// TIA Portal V15.1 export
// export: Created 2024-05-17T05:38:27.7675341Z, ExportSetting WithDefaults, DisplayName Totally Integrated Automation Portal, DisplayVersion V15.1 Update 5, DisplayName TIA Portal Openness, DisplayVersion V15.1 Update 5, DisplayName SINAMICS Startdrive Advanced, DisplayVersion V15.1, DisplayName G130, G150, S120, S150, SINAMICS MV, S210, DisplayVersion V15.1, DisplayName G110M, G120, G120C, G120D, G120P, DisplayVersion V15.1, DisplayName STEP 7 Professional, DisplayVersion V15.1 Update 5, DisplayName STEP 7 Safety, DisplayVersion V15.1, DisplayName WinCC Professional, DisplayVersion V15.1 Update 5, DisplayName SIMATIC Visualization Architect, DisplayVersion V15.1
FUNCTION "CommStnS7Sv" : Void   // FC1900, FBD
TITLE = CommStnS7Sv
{ S7_Optimized_Access := 'TRUE' }
VERSION : 0.1
// This FC sends and receives data from and to the supervision.
// stored: AutoNumber false, IsIECCheckEnabled false, SetENOAutomatically False, UDAEnableTagReadback false
   VAR_INPUT
      PlcActiveShift : Int;
      PlcActiveBreak : Int;
      AlarmA : Bool;
      AlarmB : Bool;
      AlarmC : Bool;
      AlarmD : Bool;
      ModeAutoStep : Bool;
      ModeAutoSel : Bool;
      ModeMan : Bool;
      ModeManSel : Bool;
      StnAux01Feedback_Int : Int;
      StnAux02Feedback_Int : Int;
      StnAux03Feedback_Int : Int;
      StnAux04Feedback_Int : Int;
      StnAux05Feedback_Int : Int;
      StnAux06Feedback_Int : Int;
      StnAux07Feedback_DInt : DInt;
      StnAux08Feedback_DInt : DInt;
      StnAux09Feedback_DInt : DInt;
      StnAux10Feedback_DInt : DInt;
      StnAux11Feedback_DInt : DInt;
      StnAux12Feedback_DInt : DInt;
      StnAux13Feedback_Real : Real;
      StnAux14Feedback_Real : Real;
      StnAux15Feedback_Real : Real;
      StnAux16Feedback_Real : Real;
      StnAux17Feedback_Real : Real;
      StnAux18Feedback_Real : Real;
   END_VAR
   VAR_IN_OUT
      DB_ZMToSv : "SupervisionZM";   // Send to supervision system
      DB_SvToZM : "SupervisionZM";   // Recieve from supervision system
   END_VAR
   VAR_TEMP
      Tmp_StnAux13Feedback_Real : Real;
      Tmp_StnAux14Feedback_Real : Real;
      Tmp_StnAux15Feedback_Real : Real;
      Tmp_StnAux16Feedback_Real : Real;
      Tmp_StnAux17Feedback_Real : Real;
      Tmp_StnAux18Feedback_Real : Real;
   END_VAR
BEGIN

REGION Network 1: **** 8 - Outputs **** Plc ActiveShift
   // Plc ActiveShift
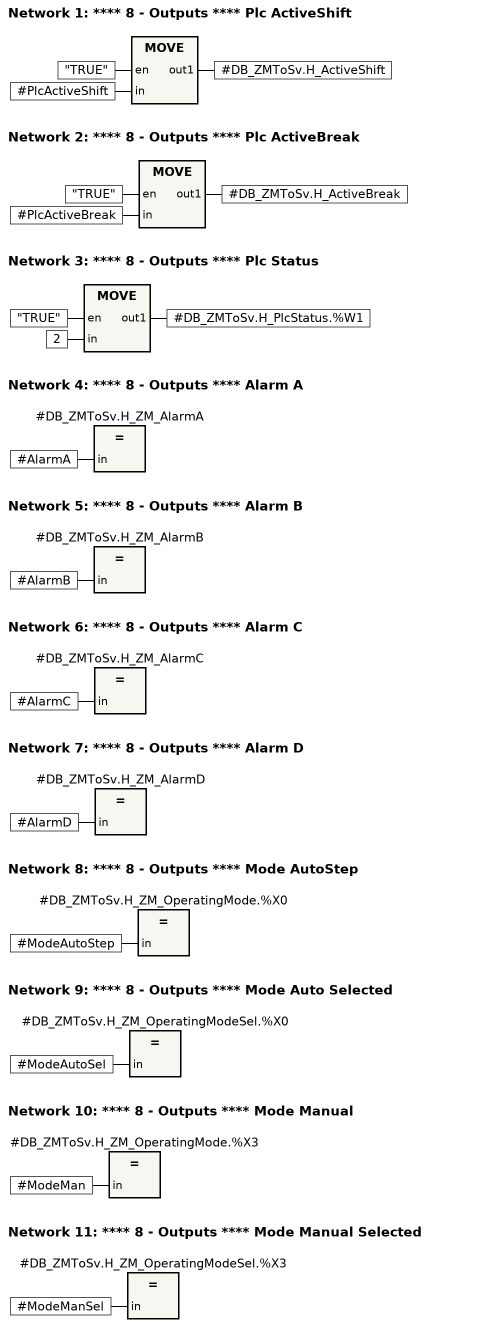
   IF "TRUE" THEN #DB_ZMToSv.H_ActiveShift := #PlcActiveShift; END_IF;
END_REGION

REGION Network 2: **** 8 - Outputs **** Plc ActiveBreak
   // Plc ActiveBreak
   IF "TRUE" THEN #DB_ZMToSv.H_ActiveBreak := #PlcActiveBreak; END_IF;
END_REGION

REGION Network 3: **** 8 - Outputs **** Plc Status
   // Plc Status
   IF "TRUE" THEN #DB_ZMToSv.H_PlcStatus.%W1 := 2; END_IF;
END_REGION

REGION Network 4: **** 8 - Outputs **** Alarm A
   // Alarm A
   #DB_ZMToSv.H_ZM_AlarmA := #AlarmA;
END_REGION

REGION Network 5: **** 8 - Outputs **** Alarm B
   // Alarm B
   #DB_ZMToSv.H_ZM_AlarmB := #AlarmB;
END_REGION

REGION Network 6: **** 8 - Outputs **** Alarm C
   // Alarm C
   #DB_ZMToSv.H_ZM_AlarmC := #AlarmC;
END_REGION

REGION Network 7: **** 8 - Outputs **** Alarm D
   // Alarm D
   #DB_ZMToSv.H_ZM_AlarmD := #AlarmD;
END_REGION

REGION Network 8: **** 8 - Outputs **** Mode AutoStep
   // Mode AutoStep
   #DB_ZMToSv.H_ZM_OperatingMode.%X0 := #ModeAutoStep;
END_REGION

REGION Network 9: **** 8 - Outputs **** Mode Auto Selected
   // Mode Auto Selected
   #DB_ZMToSv.H_ZM_OperatingModeSel.%X0 := #ModeAutoSel;
END_REGION

REGION Network 10: **** 8 - Outputs **** Mode Manual
   // Mode Manual
   #DB_ZMToSv.H_ZM_OperatingMode.%X3 := #ModeMan;
END_REGION

REGION Network 11: **** 8 - Outputs **** Mode Manual Selected
   // Mode Manual Selected
   #DB_ZMToSv.H_ZM_OperatingModeSel.%X3 := #ModeManSel;
END_REGION

REGION Network 12: **** 8 - Outputs **** Station Aux 01 Feedback
   // Station Aux 01 Feedback
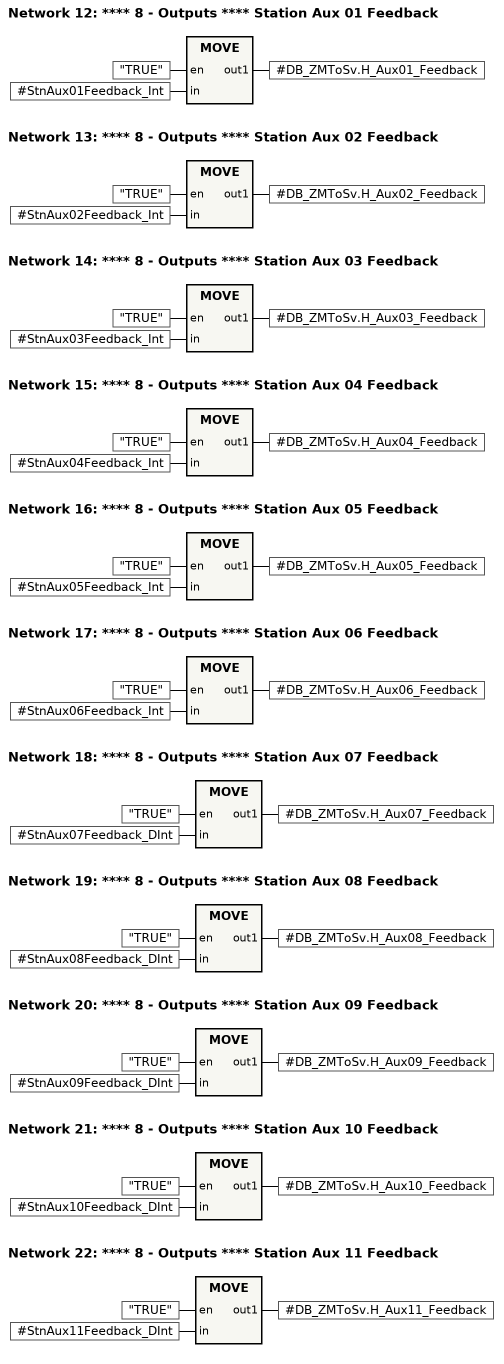
   IF "TRUE" THEN #DB_ZMToSv.H_Aux01_Feedback := #StnAux01Feedback_Int; END_IF;
END_REGION

REGION Network 13: **** 8 - Outputs **** Station Aux 02 Feedback
   // Station Aux 02 Feedback
   IF "TRUE" THEN #DB_ZMToSv.H_Aux02_Feedback := #StnAux02Feedback_Int; END_IF;
END_REGION

REGION Network 14: **** 8 - Outputs **** Station Aux 03 Feedback
   // Station Aux 03 Feedback
   IF "TRUE" THEN #DB_ZMToSv.H_Aux03_Feedback := #StnAux03Feedback_Int; END_IF;
END_REGION

REGION Network 15: **** 8 - Outputs **** Station Aux 04 Feedback
   // Station Aux 04 Feedback
   IF "TRUE" THEN #DB_ZMToSv.H_Aux04_Feedback := #StnAux04Feedback_Int; END_IF;
END_REGION

REGION Network 16: **** 8 - Outputs **** Station Aux 05 Feedback
   // Station Aux 05 Feedback
   IF "TRUE" THEN #DB_ZMToSv.H_Aux05_Feedback := #StnAux05Feedback_Int; END_IF;
END_REGION

REGION Network 17: **** 8 - Outputs **** Station Aux 06 Feedback
   // Station Aux 06 Feedback
   IF "TRUE" THEN #DB_ZMToSv.H_Aux06_Feedback := #StnAux06Feedback_Int; END_IF;
END_REGION

REGION Network 18: **** 8 - Outputs **** Station Aux 07 Feedback
   // Station Aux 07 Feedback
   IF "TRUE" THEN #DB_ZMToSv.H_Aux07_Feedback := #StnAux07Feedback_DInt; END_IF;
END_REGION

REGION Network 19: **** 8 - Outputs **** Station Aux 08 Feedback
   // Station Aux 08 Feedback
   IF "TRUE" THEN #DB_ZMToSv.H_Aux08_Feedback := #StnAux08Feedback_DInt; END_IF;
END_REGION

REGION Network 20: **** 8 - Outputs **** Station Aux 09 Feedback
   // Station Aux 09 Feedback
   IF "TRUE" THEN #DB_ZMToSv.H_Aux09_Feedback := #StnAux09Feedback_DInt; END_IF;
END_REGION

REGION Network 21: **** 8 - Outputs **** Station Aux 10 Feedback
   // Station Aux 10 Feedback
   IF "TRUE" THEN #DB_ZMToSv.H_Aux10_Feedback := #StnAux10Feedback_DInt; END_IF;
END_REGION

REGION Network 22: **** 8 - Outputs **** Station Aux 11 Feedback
   // Station Aux 11 Feedback
   IF "TRUE" THEN #DB_ZMToSv.H_Aux11_Feedback := #StnAux11Feedback_DInt; END_IF;
END_REGION

REGION Network 23: **** 8 - Outputs **** Station Aux 12 Feedback
   // Station Aux 12 Feedback
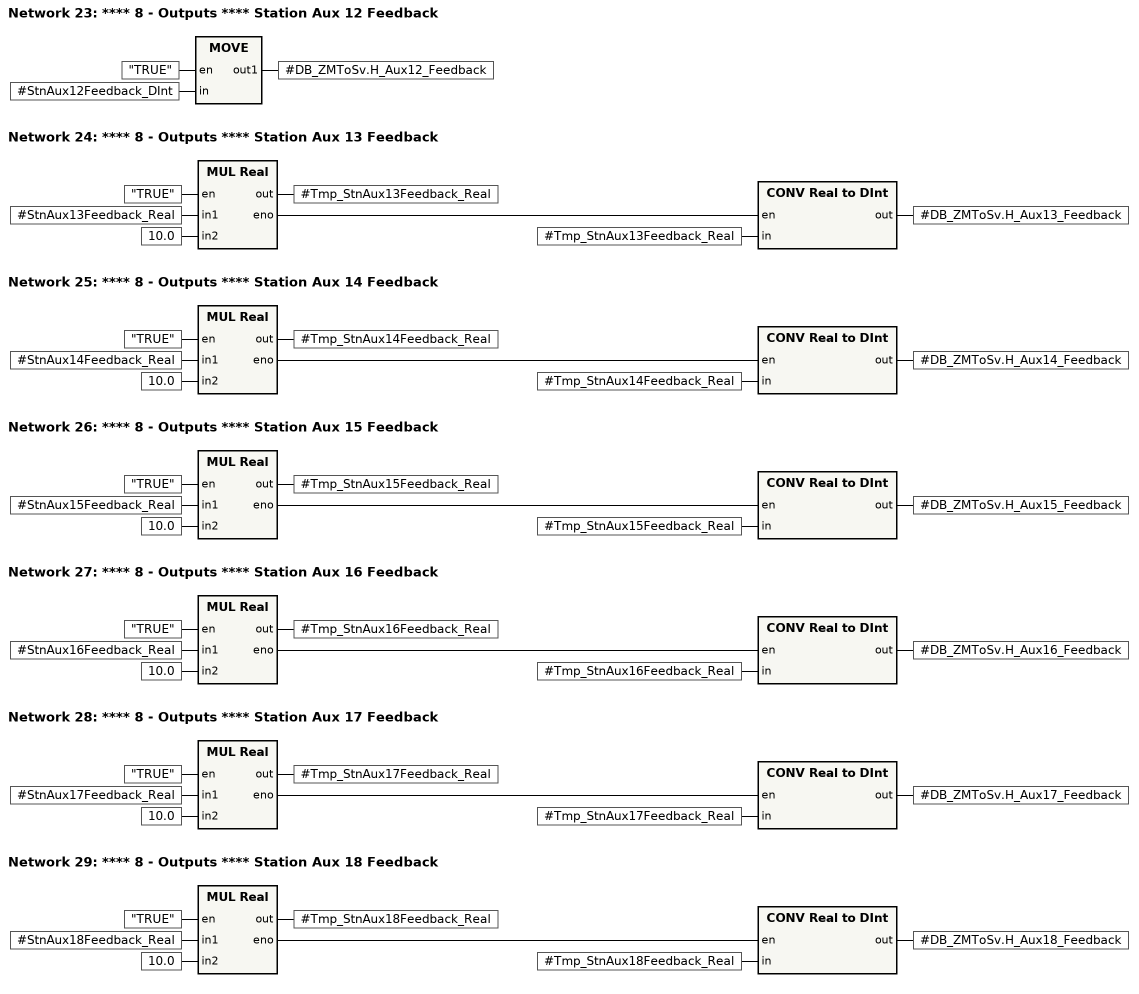
   IF "TRUE" THEN #DB_ZMToSv.H_Aux12_Feedback := #StnAux12Feedback_DInt; END_IF;
END_REGION

REGION Network 24: **** 8 - Outputs **** Station Aux 13 Feedback
   // Station Aux 13 Feedback
   IF "TRUE" THEN
       #Tmp_StnAux13Feedback_Real := #StnAux13Feedback_Real * 10.0;
       #DB_ZMToSv.H_Aux13_Feedback := REAL_TO_DINT(#Tmp_StnAux13Feedback_Real);
   END_IF;
END_REGION

REGION Network 25: **** 8 - Outputs **** Station Aux 14 Feedback
   // Station Aux 14 Feedback
   IF "TRUE" THEN
       #Tmp_StnAux14Feedback_Real := #StnAux14Feedback_Real * 10.0;
       #DB_ZMToSv.H_Aux14_Feedback := REAL_TO_DINT(#Tmp_StnAux14Feedback_Real);
   END_IF;
END_REGION

REGION Network 26: **** 8 - Outputs **** Station Aux 15 Feedback
   // Station Aux 15 Feedback
   IF "TRUE" THEN
       #Tmp_StnAux15Feedback_Real := #StnAux15Feedback_Real * 10.0;
       #DB_ZMToSv.H_Aux15_Feedback := REAL_TO_DINT(#Tmp_StnAux15Feedback_Real);
   END_IF;
END_REGION

REGION Network 27: **** 8 - Outputs **** Station Aux 16 Feedback
   // Station Aux 16 Feedback
   IF "TRUE" THEN
       #Tmp_StnAux16Feedback_Real := #StnAux16Feedback_Real * 10.0;
       #DB_ZMToSv.H_Aux16_Feedback := REAL_TO_DINT(#Tmp_StnAux16Feedback_Real);
   END_IF;
END_REGION

REGION Network 28: **** 8 - Outputs **** Station Aux 17 Feedback
   // Station Aux 17 Feedback
   IF "TRUE" THEN
       #Tmp_StnAux17Feedback_Real := #StnAux17Feedback_Real * 10.0;
       #DB_ZMToSv.H_Aux17_Feedback := REAL_TO_DINT(#Tmp_StnAux17Feedback_Real);
   END_IF;
END_REGION

REGION Network 29: **** 8 - Outputs **** Station Aux 18 Feedback
   // Station Aux 18 Feedback
   IF "TRUE" THEN
       #Tmp_StnAux18Feedback_Real := #StnAux18Feedback_Real * 10.0;
       #DB_ZMToSv.H_Aux18_Feedback := REAL_TO_DINT(#Tmp_StnAux18Feedback_Real);
   END_IF;
END_REGION
END_FUNCTION
